// Mitsubishi GX Works2 project: De07   PLC: FX2N/FX2NC

PROGRAM MAIN
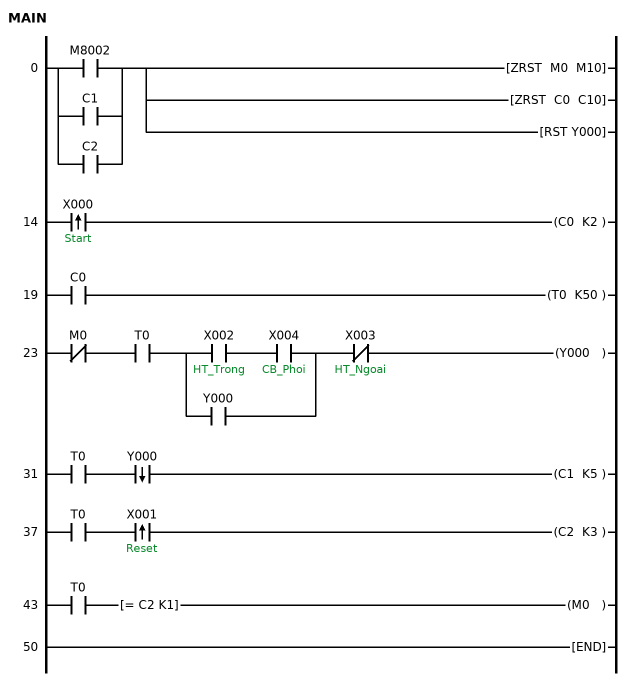
0     LD      M8002
      OR      C1
      OR      C2
      ZRST    M0 M10
      ZRST    C0 C10
      RST     Y000
14    LDP     X000  ; Start
      OUT     C0 K2
19    LD      C0
      OUT     T0 K50
23    LDI     M0
      AND     T0
      LD      X002  ; HT_Trong
      AND     X004  ; CB_Phoi
      OR      Y000
      ANB
      ANI     X003  ; HT_Ngoai
      OUT     Y000
31    LD      T0
      ANDF    Y000
      OUT     C1 K5
37    LD      T0
      ANDP    X001  ; Reset
      OUT     C2 K3
43    LD      T0
      AND=    C2 K1
      OUT     M0
50    END
END_PROGRAM
